// TIA Portal V19 export
VAR_GLOBAL   // PLC tag table "LB306"
   LB306_Scarico_Esterno_SX_Pb_ConfermaPaccoScaricato AT %I351.2 : Bool;   // 348SH3
   LB306_Scarico_Esterno_SX_Pb_Aux2 AT %I351.1 : Bool;   // 348SH2
   LB306_Scarico_Esterno_SX_Pb_PaccoReggiato AT %I351.0 : Bool;   // 348SH1
   LB306_Scarico_Esterno_SX_Lp_ConfermaPaccoScaricato AT %Q351.2 : Bool;   // 348SH3
   LB306_Scarico_Esterno_SX_Lp_Aux2 AT %Q351.1 : Bool;   // 348SH2
   LB306_Scarico_Esterno_SX_Lp_PaccoReggiato AT %Q351.0 : Bool;   // 348SH1
END_VAR
